PROGRAM WritePersistentData_1
VAR
	PersistentData			:FB_WritePersistentData;
END_VAR

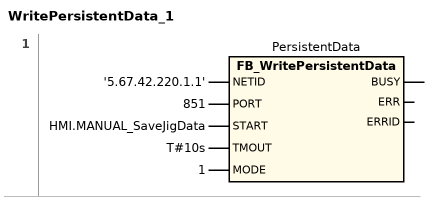
// NETWORK 1
PersistentData(
    NETID := '5.67.42.220.1.1',
    PORT := 851,
    START := HMI.MANUAL_SaveJigData,
    TMOUT := T#10s,
    MODE := 1); // FB_WritePersistentData

END_PROGRAM

(* stored: Version 1.1.0.1, ProductVersion 3.1.4024.10
   POU WritePersistentData_1: Id {7c9ae86c-8afa-4d74-8a19-e19ce9e05e10}, SpecialFunc None *)
